// Mitsubishi GX Works2 project: IELET2103_Datalab1   PLC: FX2N/FX2NC

// task Task_01 (event TRUE, interval 0, priority 31): Oppgave2_

PROGRAM Oppgave1
(* structured ladder/FBD written out as ST: instructions are called as NAME(EN, inputs, outputs); _pN, _eN, _tN stand for wires *)
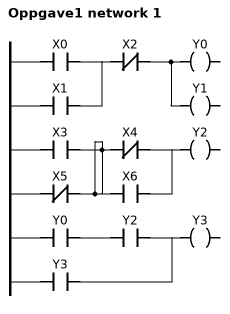
(* network 1 *)
_p1 := (X0 OR X1) AND NOT X2;
Y0 := _p1;
Y1 := _p1;
_p2 := X3 OR (NOT X5);
Y2 := (_p2 AND NOT X4) OR (_p2 AND X6);
Y3 := (Y0 AND Y2) OR Y3;
END_PROGRAM

PROGRAM Oppgave2
(* structured ladder/FBD written out as ST: instructions are called as NAME(EN, inputs, outputs); _pN, _eN, _tN stand for wires *)
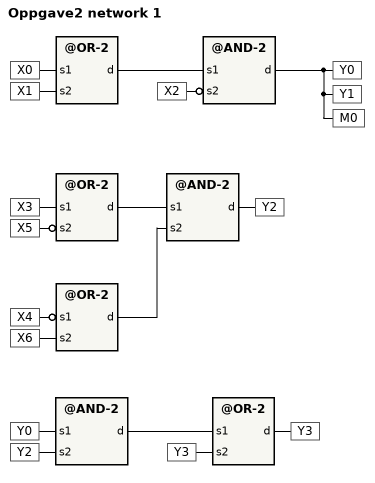
(* network 1 *)
_p1 := @AND-2(@OR-2(X0, X1), NOT X2);
Y0 := _p1;
Y1 := _p1;
M0 := _p1;
Y2 := @AND-2(@OR-2(X3, NOT X5), @OR-2(NOT X4, X6));
Y3 := @OR-2(@AND-2(Y0, Y2), Y3);
END_PROGRAM

PROGRAM Oppgave2_
END_PROGRAM
